RoboDK station: LegoLocator.rdk

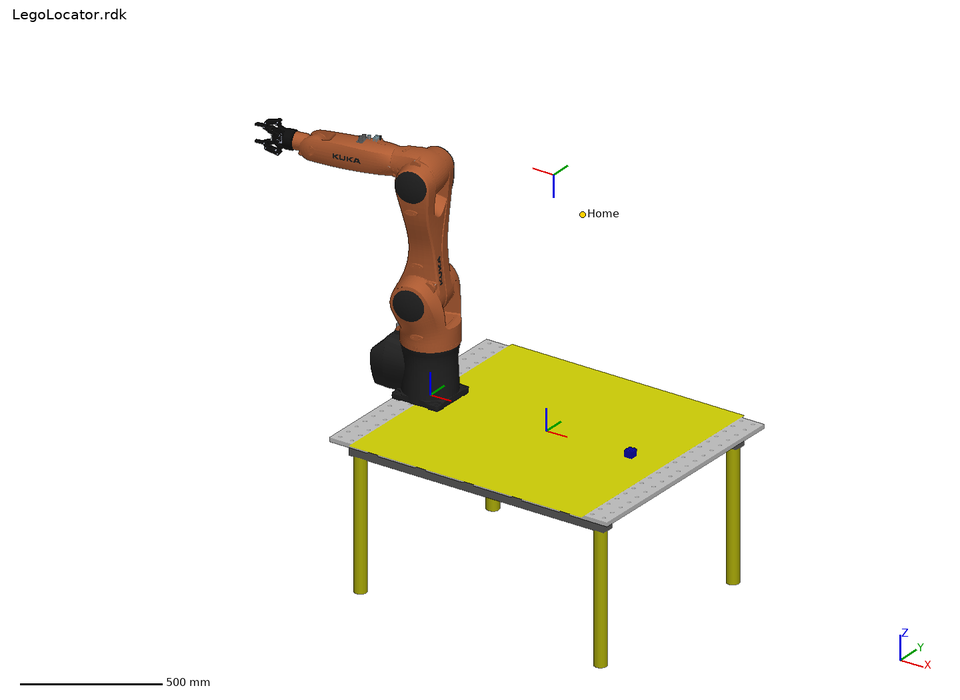
[picture v0: the station drawn from its stored meshes, robots at their saved joint values, targets as dots, program paths as lines]
Station Example-07.a-Weld Script Hexagon. Poses are relative to the parent item; angles as X-Y-Z fixed-axis rotations.
Station parameters (name, value as stored): SizeBox, 5,5,5
  - frame KUKA KR 6 R900 sixx Base at (0, 0, 0) mm
    - robot KUKA KR 6 R900 sixx: 6 axes, payload 6 kg, reach 901 mm, repeatability 0.03 mm, weight 52 kg
        modified DH rows (alpha deg, a mm, theta deg, d mm): 0, 0, 0, 400; -90, 25, 0, 0; 0, 455, -90, 0; -90, 35, 0, 420; 90, 0, 0, 0; -90, 0, 180, 80
        joint limits [-170, -190, -120, -185, -120, -350] to [170, 45, 156, 185, 120, 350]; home [0, -90, 90, 0, 0, 0]; saved at [170, -90, 90, 0, 0, 0]
      - tool Gripper RobotiQ 85 Closed, TCP at (0, 0, 130) mm, rotated rx 0 ry 90 rz 0 deg, size 134.4 x 157.6 x 75 mm
    - target Home (Cartesian target) at (655, 0, 890) mm, rotated rx 180 ry 0 rz 180 deg; joints [0, -90, 90, 0, 0, 0] of KUKA KR 6 R900 sixx
  - Python program DoWeld (listed below)
  - frame CameraRef at (530, 0, 1010) mm, rotated rx 180 ry 0 rz -180 deg
  - frame World at (500, 0, 0) mm
    - object Table at (0, 0, 0) mm, size 1193.8 x 965.2 x 609.6 mm, geometry from welding_table.sld
    - object Plane 1m x 1m at (0, 0, 0) mm, size 1000 x 1000 x 0.5 mm, geometry from plane_1m.sld
  - frame Blue at (500, 0, 0) mm
    - object Blue at (360, 0, 0) mm, size 32 x 32 x 32 mm, geometry from Blue.fbx
  - Python program Take pictures (listed below)

--- Python program DoWeld ---
from robolink import *    # API to communicate with RoboDK
from robodk import *      # robodk robotics toolbox
import cv2 as cv
import numpy as np
from matplotlib import pyplot as plt
import argparse
from numpy import loadtxt
from numpy import genfromtxt

# Any interaction with RoboDK must be done through RDK:
RDK = Robolink()
RDK.Cam2D_Close()


# get the robot by name:
robot = RDK.Item('', ITEM_TYPE_ROBOT)

# get the home target and the welding targets:
home = RDK.Item('Home')
#target = RDK.Item('Blue')

# get the pose of the target (4x4 matrix representing position and orientation):
#poseref = target.Pose()

# move the robot to home, then to the Target 1:
#robot.MoveJ(home)
#robot.MoveJ(target)
print(robot.ConnectedState())


#get the size of the lego bricks from the user
PARAM_SIZE_BOX = 'SizeBox'
SIZE_BOX = RDK.getParam('SizeBox')
size_box = RDK.getParam(PARAM_SIZE_BOX)

size_box_input = mbox('Enter the size of the box in mm [L,W,H]', entry=size_box)
if size_box_input:
    RDK.setParam(PARAM_SIZE_BOX, size_box_input)
else:
    raise Exception('Operation cancelled by user')

print(size_box_input)
robot.setJoints([180,-90,90,0,0,0])
#------------------------------------------------------------
#Select the camera and settings
cameraf=RDK.ItemUserPick('Select the Camera location (reference, tool or object)')
cam_id = RDK.Cam2D_Add(cameraf, 'FOCAL_LENGHT=6 FOV=38 FAR_LENGHT=1100 SIZE=640x480 BG_COLOR=black LIGHT_SPECULAR=white')

#-----------------------------------------------------------------------------------
#Get the height or whatever of the brick
SIZE_BOX_XYZ = [float(x.replace(' ','')) for x in SIZE_BOX.split(',')]
SIZE_BOX_Z=SIZE_BOX_XYZ[2]
#--------------------------------------------------------------------------
path= RDK.getParam('PATH_OPENSTATION')
RDK.Cam2D_Snapshot(path + "/image.png", cam_id)

imagepath=r'E:\OneDrive\OneDrive - Aalborg Universitet\AAU\8th semester\RobotVision\Miniproject\Lego\image.png'
image1=cv.imread(imagepath)

lower_color_bounds = np.array([0,100,0])
upper_color_bounds = np.array([0,255,80])

img_gray = cv.cvtColor(image1, cv.COLOR_BGR2GRAY)
mask = cv.inRange(image1,lower_color_bounds,upper_color_bounds )
mask_rgb = cv.cvtColor(mask, cv.COLOR_GRAY2BGR)
image=image1 & mask_rgb

im= cv.imread(imagepath,cv.IMREAD_GRAYSCALE)

detector=cv.SimpleBlobDetector_create()

keypoints = detector.detect(im)

im_with_keypoints=cv.drawKeypoints(im,keypoints,np.array([]),(0,0,255),cv.DRAW_MATCHES_FLAGS_DRAW_RICH_KEYPOINTS)

brick_loc=[]
for i in keypoints:
    x = i.pt[0] #i is the index of the blob you want to get the position
    y = i.pt[1]
    brick_loc.append([[x],[y],[1]])

cv.imshow("whatever",im_with_keypoints)
#mtx is the cameras intrinsic and extrinsic parameters
mtx = genfromtxt('E:\OneDrive\OneDrive - Aalborg Universitet\AAU\8th semester\RobotVision\Miniproject\Lego\mtx.csv', delimiter=',')
rvecs = genfromtxt('E:\OneDrive\OneDrive - Aalborg Universitet\AAU\8th semester\RobotVision\Miniproject\Lego\ecs.csv', delimiter=',')

print(rvecs)
print(brick_loc)




cv.waitKey()

--- Python program Take pictures ---
# Type help("robolink") or help("robodk") for more information
# Press F5 to run the script
# Documentation: https://robodk.com/doc/en/RoboDK-API.html
# Reference:     https://robodk.com/doc/en/PythonAPI/index.html
# Note: It is not required to keep a copy of this file, your python script is saved with the station
from robolink import *    # RoboDK API
from robodk import *      # Robot toolbox
RDK = Robolink()

# Notify user:
print('To edit this program:\nright click on the Python program, then, select "Edit Python script"')

# Program example:
item = RDK.Item('base')
if item.Valid():
    print('Item selected: ' + item.Name())
    print('Item posistion: ' + repr(item.Pose()))

print('Items in the station:')
itemlist = RDK.ItemList()
print(itemlist)

raise Exception('Program not edited.')
